// TIA Portal V19 export
TYPE "C701_VAR_IF_DEX_TYPIC"
   STRUCT
      TME_HOOG { ExternalAccessible := 'False'; ExternalVisible := 'False'; ExternalWritable := 'False'} : Bool;   // Ruimtetemperatuur te hoog
      STO { ExternalAccessible := 'False'; ExternalVisible := 'False'; ExternalWritable := 'False'} : Bool;   // Storing algemeen dakextractor
   END_STRUCT;
END_TYPE
